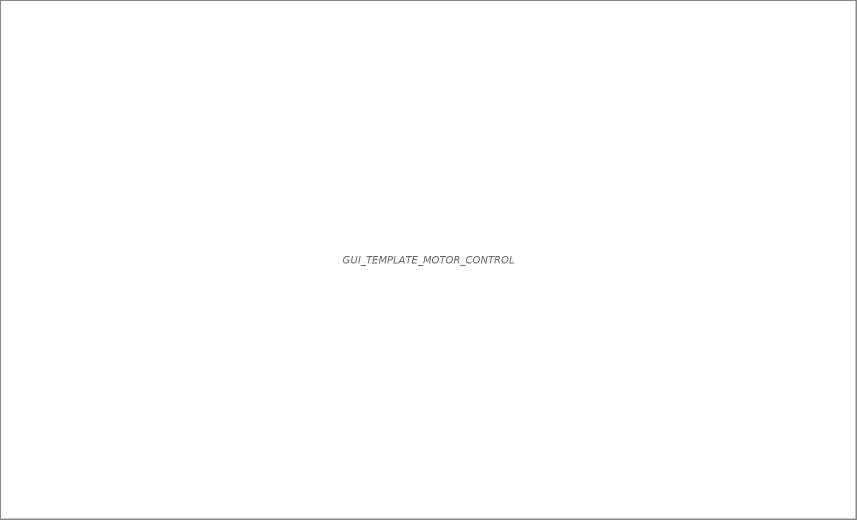
VISUALIZATION GUI_ADC_Motor2  // 857x520
    Frame (0,0 857x520)
        shows GUI_TEMPLATE_MOTOR_CONTROL(m_Instance := MAIN.adc.motor2)
END_VISUALIZATION

(* stored: Version 1.1.0.1, ProductVersion 3.1.4024.3
   Visu GUI_ADC_Motor2: Id {4db888d7-1bb4-4b40-a355-0785c845faaa} *)
